FUNCTION_BLOCK PARoutingFunction EXTENDS PAProcessFunction IMPLEMENTS IRouteableComponent
VAR_INPUT
END_VAR
VAR_OUTPUT
END_VAR
VAR
	_Points : ARRAY [1..GCL.cPointMAX] OF IACPoint;
	_PAPointMatIn1 : PAPoint(THIS^);
	_PAPointMatOut1 : PAPoint(THIS^);
END_VAR

METHOD AddPoint : BOOL
VAR_INPUT
	point : IACPoint;
END_VAR
VAR
	i: INT;
END_VAR
IF point = 0 THEN
	Addpoint := FALSE;
	RETURN;
END_IF
// 1. Check if point already exists in the array because of online change
FOR i:=1 TO GCL.cPointMAX BY 1
  DO
    IF _points[i] <> 0 THEN
		IF _points[i].ACUrl = point.ACUrl THEN
			AddPoint := FALSE;
			RETURN;			
		END_IF
	ELSE
		EXIT;
	END_IF
END_FOR;
// 2. If the point doesn't exist, add to _points-List
FOR i:=1 TO GCL.cPointMAX BY 1
  DO
    IF _points[i] = 0 THEN
		AddPoint := TRUE;
		_points[i] := point;
		EXIT;
	END_IF
END_FOR;
END_METHOD

METHOD FB_init : BOOL
VAR_INPUT
	bInitRetains : BOOL; // if TRUE, the retain variables are initialized (warm start / cold start)
	bInCopyCode : BOOL;  // if TRUE, the instance afterwards gets moved into the copy code (online change)
	parent : IACComponent;
END_VAR
AddPoint(_PAPointMatIn1);
AddPoint(_PAPointMatOut1);
END_METHOD

PROPERTY PUBLIC IsRouteStarted : BOOL
GET
VAR
	iACMethodRoute : IACMethodRouteBase;
	iControlModule : IPAControlModule;
END_VAR
IF __QUERYINTERFACE(ACMethod, iACMethodRoute) THEN
	iControlModule := iACMethodRoute.FirstCModuleInRoute;
	IF NOT (iControlModule = 0) THEN
		IF iControlModule.RoutingStateToTarget = PARoutingState.RoutePlaced THEN
			IsRouteStarted := TRUE;
			RETURN;
		END_IF		
	END_IF
END_IF
IsRouteStarted := FALSE;
END_GET
END_PROPERTY

PROPERTY PUBLIC IsRouteStopped : BOOL
GET
VAR
	iACMethodRoute : IACMethodRouteBase;
	iControlModule : IPAControlModule;
END_VAR
IF __QUERYINTERFACE(ACMethod, iACMethodRoute) THEN
	iControlModule := iACMethodRoute.LastCModuleInRoute;
	IF NOT (iControlModule = 0) THEN
		IF iControlModule.RoutingStateFromSource = PARoutingState.ReachedOffPosition THEN
			IsRouteStopped := TRUE;
			RETURN;
		END_IF		
	END_IF
END_IF
IsRouteStopped := FALSE;
END_GET
END_PROPERTY

PROPERTY PUBLIC PAPointMatIn1 : IACPoint
GET
PAPointMatIn1 := _PAPointMatIn1;
END_GET
END_PROPERTY

PROPERTY PUBLIC PAPointMatOut1 : IACPoint
GET
PAPointMatOut1 := _PAPointMatOut1;
END_GET
END_PROPERTY

PROPERTY PUBLIC Points : ARRAY [1..GCL.cPointMAX] OF IACPoint
GET
Points := _Points;
END_GET
END_PROPERTY

METHOD PROTECTED SMAborting
VAR_INPUT
END_VAR
SUPER^.SMAborting();
IF IsRouteStopped THEN
	ACState := ACStateEnum.SMAborted;
END_IF
END_METHOD

METHOD PROTECTED SMHolding
VAR_INPUT
END_VAR
SUPER^.SMHolding();
IF IsRouteStopped THEN
	ACState := ACStateEnum.SMHeld;
END_IF
END_METHOD

METHOD PROTECTED SMIdle
VAR_INPUT
END_VAR
VAR
	iACMethodRoute : IACMethodRouteBase;
END_VAR
IF  NOT(ACMethod = 0) AND __QUERYINTERFACE(ACMethod, iACMethodRoute) THEN
	iACMethodRoute.ResetRoute();
END_IF
SUPER^.SMIdle();
END_METHOD

METHOD PROTECTED SMPausing
VAR_INPUT
END_VAR
VAR
END_VAR
SUPER^.SMPausing();
IF IsRouteStopped THEN
	ACState := ACStateEnum.SMPaused;
END_IF
END_METHOD

METHOD PROTECTED SMRestarting
VAR_INPUT
END_VAR
SUPER^.SMRestarting();
IF IsRouteStarted THEN
	ACState := ACStateEnum.SMRunning;
END_IF
END_METHOD

METHOD PROTECTED SMResuming
VAR_INPUT
END_VAR
SUPER^.SMResuming();
IF IsRouteStarted THEN
	ACState := ACStateEnum.SMRunning;
END_IF
END_METHOD

METHOD PROTECTED SMRunning
VAR_INPUT
END_VAR
END_METHOD

METHOD PROTECTED SMStarting
VAR_INPUT
END_VAR
VAR
	iACMethodRoute : IACMethodRouteBase;
	route : PARoute;
END_VAR
IF __QUERYINTERFACE(ACMethod, iACMethodRoute) THEN
	
	//IF NOT iACMethodRoute.Route._IsAssigned THEN
	//	IF NOT iACMethodRoute.AssignRoute(THIS^) THEN
	//		RETURN;
	//	END_IF
	//END_IF

	route := iACMethodRoute.Route;
	IF NOT route._IsAssigned THEN
		IF NOT iACMethodRoute.AssignRoute(THIS^) THEN
			RETURN;
		END_IF
	END_IF
	
END_IF
SUPER^.SMStarting();
END_METHOD

METHOD PROTECTED SMStopping
VAR_INPUT
END_VAR
SUPER^.SMStopping();
IF IsRouteStopped THEN
	ACState := ACStateEnum.SMStopped;
END_IF
END_METHOD

END_FUNCTION_BLOCK

(* stored: Version 1.1.0.1, ProductVersion 3.1.4022.7
   POU PARoutingFunction: Id {5720e065-4c06-4434-88ae-d17ad4e83640}, SpecialFunc None
   Folder Routing: Id {a42f1ec1-22db-42b5-9c32-6ca7f38b1fce}
   Folder StateMethods: Id {d9bc5c2d-9283-4931-993b-bbcd2a63129c}
   Method AddPoint: Id {ed3f587b-2679-4903-8fa5-d2dcea533bb4}
   Method FB_init: Id {7480ef91-96bc-4fa8-a8eb-2712adb45988}
   Property IsRouteStarted: Id {929a2d8e-8761-45d6-a947-2f6b4ae1b6c0}
   Get Get: Id {cfb94747-52c2-4c9b-bcf2-7ecdbae75b43}
   Property IsRouteStopped: Id {e7a231ad-afd9-45ff-9a4f-b0efe3e454a1}
   Get Get: Id {6b5c214f-0b50-4031-b5ff-594a31d01996}
   Property PAPointMatIn1: Id {23743bf8-5b12-4f0a-bcca-02491bb9ff9d}
   Get Get: Id {40c530e2-e0e4-440a-8a7c-d26b7c890805}
   Property PAPointMatOut1: Id {8ea604cb-07ab-47b3-b19f-993275c1b91a}
   Get Get: Id {6ab608b9-d208-4467-bf45-20371cf49e48}
   Property Points: Id {272733e5-7a64-482c-8776-f6a8520a4521}
   Get Get: Id {498a4eb1-34cf-458a-9493-3b1116cd4629}
   Method SMAborting: Id {315e57f2-5654-460d-811d-4a4da64aa5a1}
   Method SMHolding: Id {2c6846d6-14b3-4a14-93b0-b600435cfdc2}
   Method SMIdle: Id {a7067a4a-7321-4df8-8868-c7e10989599a}
   Method SMPausing: Id {b679e7fa-738e-45f3-9a25-86bc4d1796f8}
   Method SMRestarting: Id {cd0e496d-086c-4ff9-9d6b-220d2018f35e}
   Method SMResuming: Id {f69a5f65-a51b-4fbb-b813-28fd68710545}
   Method SMRunning: Id {3a5e7e5a-47f4-41e9-b0da-c66f308c5330}
   Method SMStarting: Id {cf0c1bbd-2a5d-45fb-b1e5-09032a438737}
   Method SMStopping: Id {26aafd55-f14e-4a6b-9efb-6c907c1add54} *)
